FUNCTION_BLOCK FB_MOTOR
VAR_INPUT

	
END_VAR
VAR_OUTPUT
END_VAR
VAR
	z: INT;
	x : INT := 4;
	y : INT := 6 ;
END_VAR

z := x+y ;

METHOD PowerEnable : BOOL
VAR_INPUT
END_VAR
END_METHOD

END_FUNCTION_BLOCK

(* stored: Version 1.1.0.1, ProductVersion 3.1.4024.9
   POU FB_MOTOR: Id {5df450a1-b05b-432e-814f-793b25fd7bb4}, SpecialFunc None
   Method PowerEnable: Id {c98e3623-dc81-4c6d-b21e-046f5c449779} *)
